Staubli VAL3: PALLET.pjx

--- PALLET.pjx ---
Parameters version=s7.5 stackSize=5000 millimeterUnit=true
Program file=back.pgx
Program file=changeOffset.pgx
Program file=changeSpeed.pgx
Program file=computeFrame.pgx
Program file=delete.pgx
Program file=deleteItem.pgx
Program file=duplicate.pgx
Program file=find.pgx
Program file=get.pgx
Program file=getDistance.pgx
Program file=getFrame.pgx
Program file=getFrameId.pgx
Program file=getFunctionEdit.pgx
Program file=getFunctionSel.pgx
Program file=getFunctionView.pgx
Program file=getListItem.pgx
Program file=getPalletData.pgx
Program file=getPalletPos.pgx
Program file=getPoint.pgx
Program file=getSize.pgx
Program file=getSizeItem.pgx
Program file=getSizePallet.pgx
Program file=getTime.pgx
Program file=getTool.pgx
Program file=getTrajItem.pgx
Program file=getTrajType.pgx
Program file=getType.pgx
Program file=goTo.pgx
Program file=HerePoint.pgx
Program file=insertItem.pgx
Program file=load.pgx
Program file=loadAction.pgx
Program file=loadCycle.pgx
Program file=loadPage.pgx
Program file=makeTraj.pgx
Program file=new.pgx
Program file=next.pgx
Program file=onEdit.pgx
Program file=onEditItem.pgx
Program file=onEditTrsf.pgx
Program file=onFunctionEdit.pgx
Program file=onFunctionSel.pgx
Program file=onFunctionView.pgx
Program file=onInsert.pgx
Program file=onProgEnd.pgx
Program file=onRun.pgx
Program file=onSave.pgx
Program file=onStart.pgx
Program file=onStop.pgx
Program file=reset.pgx
Program file=setFrameId.pgx
Program file=setPalletData.pgx
Program file=setPalletPos.pgx
Program file=setTool.pgx
Program file=setTrajItem.pgx
Program file=showTrsf.pgx
Data file=PALLET.dtx
Library alias=saveData path=Disk://saveData/saveData.pjx
Library alias=use path=Disk://kernel/userPage/userPage.pjx
Library alias=tcp path=Disk://kernel/tool/tool.pjx
Library alias=cycleStatus path=Disk://cycleStatus/cycleStatus.pjx
Library alias=pt path=Disk://kernel/template/session/saveTraj/PALLET/PALLET.pjx
Library alias=page path=Disk://kernel/template/page/page.pjx
Library alias=language path=Disk://kernel/language/language.pjx
Library alias=language2 path=Disk://trajectory/PALLET/language/language.pjx
Type name=TrajectoryItem path=Disk://kernel/template/TrajectoryItem/TrajectoryItem.pjx
Type name=ActionItem path=Disk://kernel/template/ActionItem/ActionItem.pjx
Type name=Trajectory path=Disk://kernel/template/Trajectory/Trajectory.pjx
Type name=InstrItem path=Disk://kernel/template/InstrItem/InstrItem.pjx
Type name=TrajPallet path=Disk://kernel/template/TrajPallet/TrajPallet.pjx
Type name=FrameItem path=Disk://kernel/template/FrameItem/FrameItem.pjx
Type name=ToolItem path=Disk://kernel/template/ToolItem/ToolItem.pjx

--- PALLET.dtx ---
num nOldIndex
num nStep
string sInstruction
public string sItems
string sMessage
string sMenu
public bool bMoveType[3]
  [0] = true
  [1] = true
public bool bStepping
bool bToSave
string sTrajType
Trajectory tTraj
  [0]
    TrajectoryItem tSuper
      [0]
        num distance
        num moveType
        num nTime
        num nStop
        num nTcpAction
        string comment
        bool toStop
        mdesc nom_speed = {tmax=300, rmax=9999, leave=30, reach=30}
        InstrItem iInstr[3]
          [0]
            string sType
            string sData
          [1]
            string sType
            string sData
          [2]
            string sType
            string sData
        num nMoveId
    string sID
    num nId
mdesc mMdesc = {accel=10, vel=10, blend=off}
num nKey
frame fSetFrame = {fatherId=world[0]}
TrajPallet pEditPoint
  [0]
    TrajPointItem tData
      [0]
        TrajectoryItem tSuper
          [0]
            num distance
            num moveType
            num nTime
            num nStop
            num nTcpAction
            string comment
            bool toStop
            mdesc nom_speed = {tmax=600, rmax=9999, leave=30, reach=30}
            InstrItem iInstr[3]
              [0]
                string sType
                string sData
              [1]
                string sType
                string sData
              [2]
                string sType
                string sData
            num nMoveId
        pointRx pPoint = {fatherId=pEditPoint[0].fFrame[0]}
        num nType
    frame fFrame = {fatherId=pEditPoint[0].fReference[0]}
    num nIndexTool
    string sID
    trsf trAppro[2]
    trsf trDepart[2]
    num nX = 1
    num nY = 1
    num nZ = 1
    num nIndex
    num nDistanceXYZ[3]
      [0] = 1
      [1] = 1
      [2] = 1
    string sAction
    pointRx pO = {fatherId=pEditPoint[0].fReference[0]}
    pointRx pX = {fatherId=pEditPoint[0].fReference[0]}
    pointRx pY = {fatherId=pEditPoint[0].fReference[0]}
    pointRx pZ = {fatherId=pEditPoint[0].fReference[0]}
    num nSpeedApproach = 500
    num nSpeedDepart = 500
    num nIndexFrame
    frame fReference = {fatherId=world[0]}
string sTrajCycle

--- back.pgx ---
public program back(string x_sItem)
  local num l_nValue
  local num l_nSize
begin
  // get the value
  call getPalletPos(x_sItem,l_nValue)
  call getSizePallet(x_sItem,l_nSize)
  // set the value -1
  if l_nValue>0
    call setPalletPos(x_sItem,l_nValue-1)
  else
    call setPalletPos(x_sItem,l_nSize-1)
  endIf
end

--- changeOffset.pgx ---
public program changeOffset(num& x_nOffset[])
  local num x
  local num y
  local num z
  local point l_pPoint
  local num l_nIndex
begin
  //
  // build the pallet
  //
  // compute
  for z=0 to pEditPoint.nZ-1
    for y=0 to pEditPoint.nY-1
      for x=0 to pEditPoint.nX-1
        // set all the points
        l_pPoint=pEditPoint.tData[l_nIndex].pPoint
        l_pPoint.trsf.x=l_pPoint.trsf.x+x_nOffset*x
        l_pPoint.trsf.y=l_pPoint.trsf.y+x_nOffset[1]*y
        l_pPoint.trsf.z=l_pPoint.trsf.z+x_nOffset[2]*z
        pEditPoint.tData[l_nIndex].pPoint=l_pPoint
        l_nIndex=l_nIndex+1
      endFor
    endFor
  endFor
  //
end

--- changeSpeed.pgx ---
program changeSpeed(num x_nType, num x_nIndex)
  local string l_sMessage[2]
  local num l_nActual
  local num l_nOldValue
  local num l_nSize
  local num i
begin
  //
  // change all the speed
  //
  switch x_nType
    case 0
      // APPROACH
      call language2:message(l_sMessage,0)
      call language2:message(l_sMessage[1],2)
      l_nActual=l_nOldValue=pEditPoint.nSpeedApproach
      call use:insertDialog(l_sMessage+" "+l_sMessage[1],pEditPoint.nSpeedApproach,1,6000)
    break
    case 1
      // DEPART
      call language2:message(l_sMessage,1)
      call language2:message(l_sMessage[1],2)
      l_nActual=l_nOldValue=pEditPoint.nSpeedDepart
      call use:insertDialog(l_sMessage+" "+l_sMessage[1],pEditPoint.nSpeedDepart,1,6000)
    break
    case 2
      // NORMAL SPEED
      call language:message(l_sMessage,161)
      if pEditPoint.tData[x_nIndex].tSuper.moveType==0
        l_nActual=l_nOldValue=pEditPoint.tData[x_nIndex].tSuper.nom_speed.vel
        call use:insertDialog(l_sMessage,l_nActual,1,400)
      else
        if pEditPoint.tData[x_nIndex].tSuper.moveType==1
          l_nActual=l_nOldValue=pEditPoint.tData[x_nIndex].tSuper.nom_speed.tvel
          call use:insertDialog(l_sMessage,l_nActual,1,6000)
        endIf
      endIf
    break
  endSwitch
  // set all the speed
  if l_nActual!=l_nOldValue and x_nType==2
    // normal speed, 2
    call getSizeItem(false,l_nSize)
    for i=0 to (l_nSize-1)
      if (pEditPoint.tData[i].tSuper.moveType==0)and(l_nOldValue==pEditPoint.tData[i].tSuper.nom_speed.vel)
        pEditPoint.tData[i].tSuper.nom_speed.vel=l_nActual
      else
        if (pEditPoint.tData[i].tSuper.moveType==1)and(l_nOldValue==pEditPoint.tData[i].tSuper.nom_speed.tvel)
          pEditPoint.tData[i].tSuper.nom_speed.tvel=l_nActual
        endIf
      endIf
    endFor
  endIf
  // to be saved
  bToSave=true
end

--- computeFrame.pgx ---
public program computeFrame(num x_nNewFrame)
  local num i
begin
  // recompute all the point into the new frame
  //
  for i=0 to size(pEditPoint.tData)-1
    pEditPoint.tData[i].pPoint.trsf=!pEditPoint.tData[i].pPoint.trsf*!pEditPoint.fFrame.trsf*!pEditPoint.fReference.trsf*saveData:fFrameItem[x_nNewFrame].fFrame.trsf*pEditPoint.fFrame.trsf
  endFor
  // update the reference FRAME
  pEditPoint.fReference.trsf=saveData:fFrameItem[x_nNewFrame].fFrame.trsf
end

--- deleteItem.pgx ---
public program deleteItem(num& x_nIndex)
  local num i
  local string l_sItem
begin
  // delete the selected item
  if pEditPoint.tData[x_nIndex].nType!=1 and size(pEditPoint.tData)>3
    // delete all the field
    delete(pEditPoint.tData[x_nIndex])
  else
    // not possible to delete the point
    if  pEditPoint.tData[x_nIndex].nType!=1
      pEditPoint.tData[x_nIndex].pPoint.trsf={0,0,0,0,0,0}
    endIf
    x_nIndex=-1
  endIf
end

--- duplicate.pgx ---
public program duplicate(string x_sCopy, string x_sPaste, num& x_nResult[])
  local num i
  local num l_nSize
  local string l_sItem
  local bool l_bFound
  local num l_nResult
  local string l_sString
  local num l_nX
  local num l_nY
begin
  // duplicate

  // look if the items exist
  if insert(pt:tTraj[x_sPaste])
    // link the point
    call pt:copy_it(x_sCopy,x_sPaste)
    call pt:link_all(x_sPaste)
    // save it
    bToSave=true
  endIf
end

--- get.pgx ---
public program get(string& x_sItem[], num x_nIndex)
  local string l_sKey
  local num i
  local string l_sItem
begin
  // start from the first
  l_sKey=first(pt:tTraj)
  // search it
  while l_sKey!=""
    x_sItem=l_sKey
    l_sKey=next(pt:tTraj[l_sKey])
    if i==x_nIndex
      return
    else
      i=i+1
    endIf
  endWhile
end

--- getDistance.pgx ---
public program getDistance(tool x_tTool, num& x_nDistance[], bool x_bCycle, num x_nIndex)
  local num l_nDistance
  local point l_pPoint
  local num l_nValue
  local trsf l_trsfEmpty
  local point l_pActual
  local point l_pPrev
begin
  // first point
  if x_bCycle
    // an other one
    //
    // get the point
    //
    l_pActual=pt:tTraj[sTrajCycle].tData[x_nIndex].pPoint
    // point
    x_nDistance=distance(l_pActual.trsf,pt:tTraj[sTrajCycle].trAppro[1])
  else
    l_pActual=pEditPoint.tData[x_nIndex].pPoint
    // point
    x_nDistance=distance(l_pActual.trsf,pt:tTraj[sTrajCycle].trDepart[1])
  endIf
end

--- getFrame.pgx ---
public program getFrame(frame& x_fFrame[], bool x_bCycle)
begin
  if x_bCycle
    x_fFrame.trsf=position(pt:tTraj[sTrajCycle].fFrame,world)
  else
    // update the frame
    x_fFrame.trsf=position(pEditPoint.fFrame,world)
  endIf
end

--- getFunctionEdit.pgx ---
public program getFunctionEdit(string& x_sName[])
  local string l_sMessage
begin
  //
  // define your message for the
  // function KEY
  //
  // NOTE is an ARRAY[0..7]
  //
  // example:
  // x_sName[1]="DEMO"
  // active the F2 button
  //
  // HERE
  call language:message(l_sMessage,150)
  x_sName[0]=l_sMessage
  // ALIGN
  call language:message(l_sMessage,134)
  x_sName[1]=l_sMessage
  // REACH
  call language:message(l_sMessage,152)
  x_sName[2]=l_sMessage
  // APPROACH
  call language2:message(l_sMessage,5)
  x_sName[5]=l_sMessage
  //x_sName[5]=" "
  // DEPART
  call language2:message(l_sMessage,6)
  x_sName[6]=l_sMessage
  //x_sName[6]=" "
end

--- getFunctionView.pgx ---
public program getFunctionView(string& x_sName[])
  local string l_sMessage
begin
  //
  // define your message for the
  // function KEY
  //
  // NOTE is an ARRAY[0..7]
  //
  // example:
  // x_sName[1]="DEMO"
  // active the F2 button

  // HERE
  call language:message(l_sMessage,150)
  x_sName[0]=l_sMessage
  // ALIGN
  call language:message(l_sMessage,134)
  x_sName[1]=l_sMessage
  //
  // DISABLE
  //
  // Paste
  x_sName[3]=" "
  // Mark
  x_sName[4]=" "
  // Insert
  x_sName[5]=" "
  // Delete
  x_sName[6]=" "
end

--- getListItem.pgx ---
public program getListItem(string& x_sItem[], num x_nIndex)
  local string l_sItem[12]
  local trsf l_tTrsf
  local string l_sMessage[2]
  local point l_pPoint[2]
begin
  l_pPoint=pEditPoint.tData[x_nIndex].pPoint
  l_tTrsf=l_pPoint.trsf
  l_sItem[0]=("coord  X > "+toString(".2",l_tTrsf.x))
  l_sItem[1]=("coord  Y > "+toString(".2",l_tTrsf.y))
  l_sItem[2]=("coord  Z > "+toString(".2",l_tTrsf.z))
  l_sItem[3]=("coord RX > "+toString(".2",l_tTrsf.rx))
  l_sItem[4]=("coord RY > "+toString(".2",l_tTrsf.ry))
  l_sItem[5]=("coord RZ > "+toString(".2",l_tTrsf.rz))
  // approach
  call language2:message(l_sMessage,3)
  call use:strfill(l_sMessage,8,l_sMessage)
  call showTrsf(pEditPoint.trAppro,l_sMessage[1])
  l_sItem[6]=(l_sMessage+"1>"+l_sMessage[1])
  call showTrsf(pEditPoint.trAppro[1],l_sMessage[1])
  l_sItem[7]=(l_sMessage+"2>"+l_sMessage[1])
  // approach speed
  call language2:message(l_sMessage,5)
  call use:strfill(l_sMessage,9,l_sMessage)
  l_sItem[8]=(l_sMessage+"> "+toString("",pEditPoint.nSpeedApproach))
  // depart
  call language2:message(l_sMessage,4)
  call use:strfill(l_sMessage,8,l_sMessage)
  call showTrsf(pEditPoint.trDepart,l_sMessage[1])
  l_sItem[9]=(l_sMessage+"1>"+l_sMessage[1])
  call showTrsf(pEditPoint.trDepart[1],l_sMessage[1])
  l_sItem[10]=(l_sMessage+"2>"+l_sMessage[1])
  // depart speed
  call language2:message(l_sMessage,6)
  call use:strfill(l_sMessage,9,l_sMessage)
  l_sItem[11]=(l_sMessage+"> "+toString("",pEditPoint.nSpeedDepart))
  // copy it
  call use:stringCopy(l_sItem,x_sItem)
end

--- getPalletData.pgx ---
public program getPalletData(bool x_bCycle, TrajPallet& x_tTrajPallet)
begin
  // get the Pallet DATA
  if x_bCycle
    x_tTrajPallet=pt:tTraj[sTrajCycle]
  else
    x_tTrajPallet=pEditPoint
  endIf
end

--- getPalletPos.pgx ---
public program getPalletPos(string x_sItem, num& x_nIndex[])
  local num i
  local string l_sName
  local num l_nPos
  local num l_nSize
begin
  // init the index
  x_nIndex=-1
  // scan it
  if isDefined(pt:tTraj[x_sItem])
    x_nIndex=pt:tTraj[x_sItem].nIndex
    //
  endIf
end

--- getPoint.pgx ---
public program getPoint(point& x_pPoint[], bool x_bCycle, num x_nIndex)
  local string l_sItem
begin
  // take
  if x_bCycle
    x_pPoint=pt:tTraj[sTrajCycle].tData[x_nIndex].pPoint
  else
    // give back the point
    x_pPoint=pEditPoint.tData[x_nIndex].pPoint
  endIf
end

--- getSize.pgx ---
public program getSize(num& x_nSize[])
  local string l_sType
  local string l_sKey
  local num i
  local string l_sItem
  local string l_sPath
  local num l_nResult
begin
  // give back the size
  x_nSize=size(pt:tTraj)
end

--- getSizePallet.pgx ---
public program getSizePallet(string x_sItem, num& x_nSize)
  local string l_sType
  local string l_sKey
  local num i
begin
  //
  // get the size of the collection
  //
  if isDefined(pt:tTraj[x_sItem])
    x_nSize=size(pt:tTraj[x_sItem].tData)
  else
    x_nSize=0
  endIf
end

--- getTool.pgx ---
public program getTool(num& x_nTool)
begin
  // edit one
  x_nTool=pEditPoint.nIndexTool
end

--- getTrajItem.pgx ---
public program getTrajItem(TrajectoryItem& x_tTraj[], num x_nIndex)
begin
  //
  // get all the FIELD
  //
  x_tTraj=pEditPoint.tData[x_nIndex].tSuper
end

--- getTrajType.pgx ---
program getTrajType(string& x_sTrajType[])
  local num l_nPos
  local string l_sPath
begin
  // get the trajType
  l_sPath=libPath()
  if find(l_sPath,sTrajType)==-1 or sTrajType==""
    do
      l_nPos=find(l_sPath,"/")
      if l_nPos==-1
        l_nPos=find(l_sPath,"\")
      endIf
      if l_nPos!=-1
        l_sPath=right(l_sPath,len(l_sPath)-l_nPos-1)
      endIf
    until l_nPos==-1
    //
    sTrajType=l_sPath
  endIf
  // return back
  x_sTrajType=sTrajType
end

--- getType.pgx ---
public program getType(num& x_nType, bool x_bCycle, num x_nIndex)
begin
  // get the point Type
  if x_bCycle
    x_nType=pt:tTraj[sTrajCycle].tData[x_nIndex].nType
  else
    x_nType=pEditPoint.tData[x_nIndex].nType
  endIf
end

--- goTo.pgx ---
public program goTo(tool x_tTool, mdesc x_mDesc, num x_nMoveType, bool& x_bUnreached[], num x_nIndex)
  local string l_sMessage
  local num i
  local point l_pPoint
  local joint l_jJoint
begin
  // the maximum size
  x_mDesc.blend=off
  // get the point
  call getPoint(l_pPoint,false,x_nIndex)
  //
  // step by step motion
  //
  // go to the appro
  for i=0 to size(pEditPoint.trAppro)-1
    if !pointToJoint(x_tTool,herej(),appro(l_pPoint,pEditPoint.trAppro[i]),l_jJoint)
      // not reachable
      call language:message(l_sMessage,169)
      popUpMsg(l_sMessage)
      return
    else
      if x_nMoveType==0 and i==0
        // or is not in range
        movej(appro(l_pPoint,pEditPoint.trAppro[i]),x_tTool,x_mDesc)
      else
        movel(appro(l_pPoint,pEditPoint.trAppro[i]),x_tTool,x_mDesc)
      endIf
    endIf
  endFor
  // wait to catch the point
  wait(isEmpty() or isKeyPressed(255) or cycleStatus:nWorkingStatus!=0)
  if isEmpty()
    delay(1)
    // go directly to the point is the robot is nearby the point
    if !pointToJoint(x_tTool,herej(),l_pPoint,l_jJoint)
      // not reachable
      call language:message(l_sMessage,169)
      popUpMsg(l_sMessage)
      return
    else
      movel(l_pPoint,x_tTool,x_mDesc)
      wait(isEmpty() or isKeyPressed(255) or cycleStatus:nWorkingStatus!=0)
      if isEmpty()
        delay(1)
        // go to the depart
        for i=0 to size(pEditPoint.trDepart)-1
          if !pointToJoint(x_tTool,herej(),appro(l_pPoint,pEditPoint.trDepart[i]),l_jJoint)
            // not reachable
            call language:message(l_sMessage,169)
            popUpMsg(l_sMessage)
            return
          else
            movel(appro(l_pPoint,pEditPoint.trDepart[i]),x_tTool,x_mDesc)
          endIf
        endFor
        wait(isEmpty() or isKeyPressed(255) or cycleStatus:nWorkingStatus!=0)
      endIf
    endIf
  endIf
end

--- HerePoint.pgx ---
public program HerePoint(num x_nIndex)
  local tool l_tTool
  local point l_pHere
  local frame l_fFrame
  local num i
  local num l_nIndex
  local num l_nSize
begin
  //
  // take the point
  //
  // tool
  call tcp:getTool(l_tTool,pEditPoint.nIndexTool)
  // here
  l_pHere=here(l_tTool,pEditPoint.fFrame)
  resetMotion()
  // save the trsf
  pEditPoint.tData[x_nIndex].pPoint.trsf=l_pHere.trsf
  // check the moveType to save the config
  if pEditPoint.tData[x_nIndex].tSuper.moveType==0
    pEditPoint.tData[x_nIndex].pPoint.config=l_pHere.config
  endIf
end

--- insertItem.pgx ---
public program insertItem(num& x_nIndexCopy, num x_nIndexPaste)
  local num l_nLastType
  local point l_pPoint
  local num l_nType
begin
  //
  // use to add more elements from the typical one
  //
  // insert all the field
  //
  l_pPoint=pEditPoint.tData[x_nIndexCopy].pPoint
  link(pEditPoint.tData[x_nIndexPaste].pPoint,pEditPoint.fFrame)
  insert(pEditPoint.tData[x_nIndexPaste])
  // set IT
  pEditPoint.tData[x_nIndexPaste].pPoint.trsf=l_pPoint.trsf
end

--- load.pgx ---
public program load(string x_sItem, num& x_nResult)
  local string l_sType
  local string l_sMessage
  local num i
  local num l_nResult
begin
  // load the select trajectory..already loaded
  call getTrajType(l_sType)
  if find(pt:libPath(),saveData:sPathTraj)==-1
    l_nResult=pt:libLoad(saveData:sPathTraj+l_sType)
    delay(0)
    if saveData:bDebug or l_nResult!=0
      ? "loading PALLET..."+saveData:sPathTraj+l_sType + toString("",l_nResult)
    endIf
  endIf
  // use the type...
  if isDefined(pt:tTraj[x_sItem])
    call pt:link_all(x_sItem)
    pEditPoint=pt:tTraj[x_sItem]
    pEditPoint.sID=x_sItem
    link(pEditPoint.fReference,world)
    link(pEditPoint.fFrame,pEditPoint.fReference)
  elseIf x_sItem!=""
    // not FOUND
    call language:message(l_sMessage,-7)
    x_nResult=-1
    popUpMsg(l_sMessage+x_sItem)
    pEditPoint.sID=""
  endIf
end

--- loadAction.pgx ---
program loadAction(string x_sPallet, num x_nOffset)
  local num l_nPos
  local num l_nSize[3]
  local string l_sAction
begin
  //
  // get the actual position
  //
  call getPalletPos(x_sPallet,l_nPos)
  // PLANE CONDITION
  // loook for the z quote
  l_sAction=pt:tTraj[sTrajCycle].sAction[l_nPos%pt:tTraj[sTrajCycle].nZ]
  if (l_nPos+1)%(pt:tTraj[sTrajCycle].nY*pt:tTraj[sTrajCycle].nX)==0 and l_sAction!=""
    // show the string
    cycleStatus:sToShow="CALL PALLET PROG "+l_sAction
    // SET THE JUMP for the CALL..
    cycleStatus:bCALL=true
    // NB use the session field
    cycleStatus:iToSuperV.sType="PROG"
    cycleStatus:iToSuperV.sData=l_sAction
    use:bUseRefresh=true
  endIf
end

--- loadCycle.pgx ---
public program loadCycle(string x_sItem, num& x_nResult[])
  local string l_sType
  local string l_sMessage
begin
  // load the select trajectory..already loaded
  call getTrajType(l_sType)
  if find(pt:libPath(),saveData:sPathTraj)==-1
    pt:libLoad(saveData:sPathTraj+l_sType)
    delay(0)
    if saveData:bDebug
      ? "loading PALLET..."+saveData:sPathTraj+l_sType
    endIf
  endIf
  if isDefined(pt:tTraj[x_sItem])
    call pt:link_all(x_sItem)
    // use the type...
    sTrajCycle=x_sItem
  else
    // not FOUND
    call language:message(l_sMessage,-7)
    x_nResult=-1
    cycleStatus:bToStop=true
    popUpMsg(l_sMessage+x_sItem)
  endIf
end

--- loadPage.pgx ---
program loadPage(string x_sPage, string& x_sItems[])
// load the next page
  local num i
  local string l_sMessage
begin
  // look if the page libload is correct
  i=page:libLoad(x_sPage)
  delay(0)
  if i!=0
    logMsg("[KERNEL] INTERFACE:PAGE LIBLOAD "+x_sPage+" result "+toString("",i))
    call language:message(l_sMessage,-7)
    popUpMsg(l_sMessage+x_sPage+" ; "+toString("",i))
  else
    // copy all the field from x_sItems to the next page
    call use:stringCopy(x_sItems,page:sItems)
    call page:main()
    // to give back
    call use:stringCopy(page:sItems,x_sItems)
  endIf
end

--- makeTraj.pgx ---
public program makeTraj(string& x_sItem[])
  local num i
  local num l_nDistance
  local num l_nSize
  local tool l_tTool
  local num l_nMoveId
  local point l_pPoint
  local string l_sType
  local TrajectoryItem l_tTraj
  local ActionItem l_aAction
  local num l_nIndex
  local mdesc l_nomSpeed
begin
  // take the TOOL
  call tcp:getTool(l_tTool,pt:tTraj[sTrajCycle].nIndexTool)
  // the maximum size
  call getSizeItem(true,l_nSize)
  //
  // for all of my traj cyclePoints move the robot
  //
  // one element
  resize(tTraj.tSuper,1,1)
  tTraj.tSuper=pt:tTraj[sTrajCycle].tData[pt:tTraj[sTrajCycle].nIndex].tSuper
  tTraj.tSuper.comment="["+toString("2",pt:tTraj[sTrajCycle].nIndex+1)+"/"+toString("2",size(pt:tTraj[sTrajCycle].tData))+"] "+tTraj.tSuper.comment
  tTraj.sID="PALLET "+pt:tTraj[sTrajCycle].sID
  call cycleStatus:addTraj(tTraj)
  //
  // get the point info
  //
  l_nIndex=pt:tTraj[sTrajCycle].nIndex
  l_tTraj=pt:tTraj[sTrajCycle].tData[l_nIndex].tSuper
  call getPoint(l_pPoint,true,l_nIndex)
  //
  // put the move in the stack
  //
  // go to the appro
  for i=0 to size(pt:tTraj[sTrajCycle].trAppro)-1
    if l_tTraj.moveType==0 and i==0
      // or is not in range
      movej(appro(l_pPoint,pt:tTraj[sTrajCycle].trAppro[i]),l_tTool,l_tTraj.nom_speed)
    elseIf i==0
      movel(appro(l_pPoint,pt:tTraj[sTrajCycle].trAppro[i]),l_tTool,l_tTraj.nom_speed)
    elseIf i>0 and pt:tTraj[sTrajCycle].trAppro[i]!=pt:tTraj[sTrajCycle].trAppro[i-1]
      l_nomSpeed=l_tTraj.nom_speed
      l_nomSpeed.tvel=pt:tTraj[sTrajCycle].nSpeedApproach
      l_nomSpeed.leave=l_nomSpeed.reach=5
      movel(appro(l_pPoint,pt:tTraj[sTrajCycle].trAppro[i]),l_tTool,l_nomSpeed)
    endIf
  endFor
  //
  // get the distance in percentage
  call getDistance(l_tTool,l_nDistance,true,l_nIndex)
  //
  // give to the traj library the percentage distance
  //
  if l_tTraj.toStop
    l_tTraj.nom_speed.blend=off
  endIf
  // send the action information to cycle
  l_tTraj.nom_speed.tvel=pt:tTraj[sTrajCycle].nSpeedDepart
  l_nMoveId=movel(l_pPoint,l_tTool,l_tTraj.nom_speed)
  l_aAction.nDistance=l_nDistance
  l_aAction.nPointId=0
  l_aAction.nMoveId=l_nMoveId
  l_aAction.sIdTraj="PALLET "+pt:tTraj[sTrajCycle].sID
  call cycleStatus:putInstr_Traj(l_aAction,l_tTraj,pt:tTraj[sTrajCycle].nIndexTool,1)
  // there is a waitEndMove
  if l_tTraj.toStop
    waitEndMove()
    delay(l_tTraj.nStop)
    // wait all the action has been done
    wait(cycleStatus:bActionRunning==false)
  endIf
  // update
  l_tTraj=pt:tTraj[sTrajCycle].tData[l_nIndex].tSuper
  //  depart
  for i=0 to size(pt:tTraj[sTrajCycle].trDepart)-1
    l_nomSpeed=l_tTraj.nom_speed
    l_nomSpeed.tvel=pt:tTraj[sTrajCycle].nSpeedDepart
    if pt:tTraj[sTrajCycle].trDepart[0]!=pt:tTraj[sTrajCycle].trDepart[1]
      l_nomSpeed.leave=l_nomSpeed.reach=5
    endIf
    movel(appro(l_pPoint,pt:tTraj[sTrajCycle].trDepart[i]),l_tTool,l_nomSpeed)
  endFor
  // calculate the offset
  l_nDistance=distance(l_pPoint,appro(l_pPoint,pt:tTraj[sTrajCycle].trDepart[i-1]))
  // use a 10 % of tollerance
  if l_nDistance!=0
    l_nDistance=1-l_tTraj.nom_speed.leave/l_nDistance-0.1
  else
    l_nDistance=1-0.1
  endIf
  //
  // ACTION AFTER MOVE
  //
  call loadAction(x_sItem,l_nDistance)
end

--- next.pgx ---
public program next(string x_sItem)
  local num l_nValue
  local num l_nSize
begin
  // get the actual position
  call getPalletPos(x_sItem,l_nValue)
  call getSizePallet(x_sItem,l_nSize)
  // go to the next ONE
  if l_nValue<l_nSize-1
    call setPalletPos(x_sItem,l_nValue+1)
  else
    call setPalletPos(x_sItem,0)
  endIf
end

--- onEdit.pgx ---
public program onEdit(string& x_sItem[])
  local string l_sPath
  local num i
  local string l_sItem
  local num l_nSize
  local num l_nResult
begin
  // DEFINE YOUR ITEM
  call getTrajType(saveData:sTrajTypeUsing)
  // load the trajectory
  call load(x_sItem,l_nResult)
  if find(x_sItem,"@")==-1
    // load the page viewTraj
    l_sPath="Disk://trajectory/PALLET/page_pallet"
    // give back the path
    x_sItem[1]=x_sItem
    x_sItem=l_sPath
  endIf
end

--- onEditItem.pgx ---
public program onEditItem(string& x_sEvent[], num x_nIndex, num x_nIndexItem)
  local bool l_bReachable
  local num i
  local trsf l_tApproach[2]
  local trsf l_tDepart[2]
  local num l_nSpeed
  local string l_sMessage
  local num l_nOffset
  local string l_sMessage2
  local string l_sItem
begin
  // edit the custom element that was add in the list
  if x_nIndex<6
    // edit the TRSF
    call onEditTrsf(x_nIndex,x_nIndexItem,x_sEvent)
  else
    // i=find(x_sEvent,">")+1
    call use:findPos(x_sEvent,">",i)
    i=i+1
    call language2:message(l_sMessage2,42)
    //
    switch x_nIndex
      case 6
        // change the approach 1
        call language2:message(l_sMessage,3)
        call use:changeTrsf(pEditPoint.trAppro,l_sMessage+" [1]",l_sMessage2)
      break
      case 7
        // change the approach 2
        call language2:message(l_sMessage,3)
        call use:changeTrsf(pEditPoint.trAppro[1],l_sMessage+" [2]",l_sMessage2)
      break
      case 8
        // change the approach speed
        call use:listcursor(use:nView,false)
        l_sItem=""
        call use:changeValue(pEditPoint.nSpeedApproach,1,2000,i+40-use:nBottomX,use:nView+1,l_sItem)
      break
      case 9
        // change the depart
        call language2:message(l_sMessage,4)
        call use:changeTrsf(pEditPoint.trDepart,l_sMessage+" [1]",l_sMessage2)
      break
      case 10
        // change the depart 2
        call language2:message(l_sMessage,4)
        call use:changeTrsf(pEditPoint.trDepart[1],l_sMessage+" [2]",l_sMessage2)
      break
      case 11
        // change the depart speed
        call use:listcursor(use:nView,false)
        l_sItem=""
        call use:changeValue(pEditPoint.nSpeedDepart,1,2000,i+40-use:nBottomX,use:nView+1,l_sItem)
      break
    endSwitch
  endIf
  //
end

--- onEditTrsf.pgx ---
public program onEditTrsf(num x_nIndex, num x_nIndexItem, string x_sEvent)
  local num i
  local num l_nMin
  local num l_nMax
  local trsf l_tTrsf
  local string l_sEmpty
  local joint l_jJoint
  local tool l_tTool
  local string l_sMessage
  local trsf l_OldTrsf
begin
  // edit TRSF OF THE POINT
  l_tTrsf=pEditPoint.tData[x_nIndexItem].pPoint.trsf
  // find the >
  call use:findPos(x_sEvent,">",i)
  i=i+1
  // find the line
  if !cycleStatus:bCycle
    l_nMin=l_nMax=0
  else
    switch x_nIndex
      case 0
        // x
        l_nMin=l_tTrsf.x-10
        l_nMax=l_tTrsf.x+10
      break
      case 1
        // y
        l_nMin=l_tTrsf.y-10
        l_nMax=l_tTrsf.y+10
      break
      case 2
        // z
        l_nMin=l_tTrsf.z-10
        l_nMax=l_tTrsf.z+10
      break
      case 3
        // rx
        l_nMin=l_tTrsf.rx-5
        l_nMax=l_tTrsf.rx+5
      break
      case 4
        // ry
        l_nMin=l_tTrsf.ry-5
        l_nMax=l_tTrsf.ry+5
      break
      case 5
        // rz
        l_nMin=l_tTrsf.rz-5
        l_nMax=l_tTrsf.rz+5
      break
    endSwitch
  endIf
  // clean the line
  call use:listcursor(use:nView,false)
  //
  switch x_nIndex
    case 0
      //  x-value
      call use:changeValue(l_tTrsf.x,l_nMin,l_nMax,i+40-use:nBottomX,use:nView+1,l_sEmpty)
    break
    case 1
      //  y-value
      call use:changeValue(l_tTrsf.y,l_nMin,l_nMax,i+40-use:nBottomX,use:nView+1,l_sEmpty)
    break
    case 2
      //  z-value
      call use:changeValue(l_tTrsf.z,l_nMin,l_nMax,i+40-use:nBottomX,use:nView+1,l_sEmpty)
    break
    case 3
      //  rx-value
      call use:changeValue(l_tTrsf.rx,l_nMin,l_nMax,i+40-use:nBottomX,use:nView+1,l_sEmpty)
    break
    case 4
      //  ry-value
      call use:changeValue(l_tTrsf.ry,l_nMin,l_nMax,i+40-use:nBottomX,use:nView+1,l_sEmpty)
    break
    case 5
      //  rz-value
      call use:changeValue(l_tTrsf.rz,l_nMin,l_nMax,i+40-use:nBottomX,use:nView+1,l_sEmpty)
    break
  endSwitch
  // validate
  if !use:bUseEscape
    // check the config
    l_tTool=saveData:tData[pEditPoint.nIndexTool].tcp
    l_OldTrsf=pEditPoint.tData[x_nIndexItem].pPoint.trsf
    pEditPoint.tData[x_nIndexItem].pPoint.trsf=l_tTrsf
    if !pointToJoint(l_tTool,herej(),pEditPoint.tData[x_nIndexItem].pPoint,l_jJoint)
      // not reachable
      pEditPoint.tData[x_nIndexItem].pPoint.trsf=l_OldTrsf
      call language:message(l_sMessage,169)
      popUpMsg(l_sMessage)
    endIf
  endIf
end

--- onFunctionEdit.pgx ---
public program onFunctionEdit(num x_nIndex, string x_sEvent, num x_nFunctionKey)
  local string l_sMessage
  local string l_sButton[2]
  local bool l_bOk
  local string l_sPage
  local string l_sItem
  local tool l_tTool
  local point l_pAlign
  local bool l_bYes
  local string l_sMessage2
begin
  //
  // do on Key action
  //
  // x_nIndex = actual index item
  // x_sEvent = actual event item
  //
  switch x_nFunctionKey
    // F1 button
    case 271
      // HERE POINT
      if !cycleStatus:bCycle
        call language:message(l_sMessage,160)
        call language:getYesNo(l_sButton)
        call use:yes_no(l_sMessage,l_sButton,l_bOk)
        if l_bOk
          call HerePoint(x_nIndex)
        endIf
      endIf
    break
    // F2 button
    case 272
      // ALIGN
      if !cycleStatus:bCycle
        resetMotion()
        call getFrame(fSetFrame,false)
        // tool
        call tcp:getTool(l_tTool,pEditPoint.nIndexTool)
        l_pAlign=here(l_tTool,world)
        l_pAlign.trsf=align(l_pAlign.trsf,fSetFrame.trsf)
        call language:message(l_sMessage,203)
        call language:message(l_sMessage2,134)
        l_sMessage=l_sMessage+" "+l_sMessage2+"..."
        call use:timerDialog(l_sMessage,0)
        movej(l_pAlign,l_tTool,mMdesc)
        watch(isEmpty() or isKeyPressed(255),3)
        if !isEmpty()
          resetMotion()
        endIf
        delay(2)
      endIf
    break
    // F3 button
    case 273
      // Select the gun
      l_sPage="Disk://kernel/page/tool"
      call loadPage(l_sPage,l_sItem)
      // set the tool
      pEditPoint.nIndexTool=saveData:nIndexTool
    break
    // F4 button
    case 274
    break
    // F5 button
    case 275
    break
    // F6 button
    case 276
      // change all the approach speed
      call changeSpeed(0,x_nIndex)
    break
    // F7 button
    case 277
      // change all the depart speed
      call changeSpeed(1,x_nIndex)
    break
    // F8 button
    case 278
      // save it
      bToSave=true
    break
  endSwitch
end

--- onFunctionSel.pgx ---
public program onFunctionSel(num x_nIndex, string x_sEvent, num x_nFunctionKey)
begin
  //
  // do on Key action
  //
  // x_nIndex = actual index item
  // x_sEvent = actual event item
  //
  switch x_nFunctionKey
    // F1 button
    case 271
    break
    // F2 button
    case 272
    break
    // F3 button
    case 273
    break
    // F4 button
    case 274
    break
    // F5 button
    case 275
    break
    // F6 button
    case 276
    break
    // F7 button
    case 277
    break
    // F8 button
    case 278
    break
  endSwitch
end

--- onFunctionView.pgx ---
public program onFunctionView(num x_nIndex, string x_sEvent, num x_nFunctionKey)
  local string l_sMessage
  local string l_sButton[2]
  local bool l_bOk
  local tool l_tTool
  local point l_pAlign
  local string l_sMessage2
  local joint l_jJoint
begin
  //
  // do on Key action
  //
  // x_nIndex = actual index item
  // x_sEvent = actual event item
  //
  switch x_nFunctionKey
    case 271
      // HERE POINT
      if !cycleStatus:bCycle
        call language:message(l_sMessage,160)
        call language:getYesNo(l_sButton)
        call use:yes_no(l_sMessage,l_sButton,l_bOk)
        if l_bOk
          call HerePoint(x_nIndex)
        endIf
      endIf
    break
    // F2 button
    case 272
      // ALIGN
      if !cycleStatus:bCycle and !cycleStatus:bSimulation
        resetMotion()
        call getFrame(fSetFrame,false)
        // tool
        call tcp:getTool(l_tTool,pEditPoint.nIndexTool)
        l_pAlign=here(l_tTool,world)
        l_pAlign.trsf=align(l_pAlign.trsf,fSetFrame.trsf)
        // check the align
        if pointToJoint(l_tTool,herej(),l_pAlign,l_jJoint)
          call language:message(l_sMessage,203)
          call language:message(l_sMessage2,134)
          l_sMessage=l_sMessage+" "+l_sMessage2+"..."
          call use:timerDialog(l_sMessage,0)
          movel(l_pAlign,l_tTool,mMdesc)
          watch(isEmpty() or isKeyPressed(255),3)
          if !isEmpty()
            resetMotion()
          endIf
          delay(2)
        endIf
      endIf
    break
    // F3 button
    case 273
    break
    // F4 button
    case 274
    break
    // F5 button
    case 275
    break
    // F6 button
    case 276
    break
    // F7 button
    case 277
    break
    // F8 button
    case 278
    break
  endSwitch
end

--- onInsert.pgx ---
public program onInsert(string& x_sItem[])
  local string l_sEvent
  local num l_nKey
  local num l_nIndex
  local num l_nSize
  local num i
  local string l_sMessage
  local bool l_bFound
  local string l_sType
  local bool l_bUseFilter
  local string l_sPaste
  local num l_nResult
  local num l_nX
  local num l_nY
  local string l_sName
begin
  // get the type
  call getTrajType(x_sItem)
  saveData:sTrajTypeUsing=x_sItem
  cls()
  // is a filter using ??
  if saveData:sTrajFilter!=""
    l_bUseFilter=true
    call language:message(l_sMessage,64)
    call use:type(0,1,l_sMessage+">ON")
  else
    // clean
    call use:typeLen(0,1," ",use:nBottomX)
  endIf
  //
  // CREATE THE LIST
  //
  // define your list size for default
  call use:setSizeList(19,0,19,11)
  call use:setView(false)
  call use:listcreate(x_sItem)
  // take the coordinate....
  l_nX=40-use:nBottomX-1
  l_nY=use:nBottomY+1
  // show the message
  call language:message(l_sMessage,61)
  call use:stringToArray(l_sMessage,sMenu)
  call use:setMenu(sMenu,true,3)
  // Build the list
  call getSize(l_nSize)
  for i=0 to l_nSize-1
    call get(l_sEvent,i)
    if l_sEvent!=""
      //
      // use the filter ?
      //
      // check if the bProcessList filter is active
      //
      l_bFound=true
      if saveData:sTrajFilter!=""
        l_bFound=find(l_sEvent,saveData:sTrajFilter)!=-1
      endIf
      // add
      if l_bFound
        call use:listadd(l_sEvent)
      endIf
    endIf
  endFor
  call use:listupdate(0)
  do
    // get the item
    l_nKey=get()
    call use:listevent(l_nKey,l_nIndex,l_sEvent)
    if l_nKey==271 and l_bUseFilter
      // Build the list
      call getSize(l_nSize)
      // empty and rebuild
      call use:listempty()
      for i=0 to l_nSize-1
        call get(l_sEvent,i)
        if l_sEvent!=""
          call use:listadd(l_sEvent)
        endIf
      endFor
      // clean
      call use:typeLen(0,1," ",use:nBottomX)
      call use:typeMenu(1," ")
      l_bUseFilter=false
      call use:listupdate(0)
    endIf
        //
  until l_nKey==270 or l_nKey==255 or l_nKey==278 or l_nKey==276
  //
  switch l_nKey
    case 270
      // save the name
      l_sName=l_sEvent
    break
    case 276
      // duplicate
      // ask for the new
      call language:message(l_sMessage,21)
      call use:type(l_nX,l_nY,l_sMessage)
      l_sName=l_sEvent
      // read the new trajectory
      call use:read(l_nX+len(l_sMessage),l_nY,l_sName,10,false)
      if !use:bUseEscape
        call duplicate(l_sEvent,l_sName,l_nResult)
      endIf
    break
    case 278
      call language:message(l_sMessage,21)
      call use:type(l_nX,l_nY,l_sMessage)
      // read the new trajectory
      call use:read(l_nX+len(l_sMessage),l_nY,l_sName,10,false)
      if !use:bUseEscape
        // look if the items exist
        call new(l_sName,l_nResult)
        if l_nResult==-1
          call language:message(l_sMessage,-2)
          popUpMsg(l_sMessage)
        endIf
      endIf
    break
  endSwitch
  if l_nKey!=255
    x_sItem=l_sName
  else
    x_sItem=""
  endIf
end

--- onRun.pgx ---
public program onRun(string& x_sItem[])
  local string l_sEmpty
  local num l_nResult
begin
  // execute check if need to reload
  call loadCycle(x_sItem,l_nResult)
  // execute
  call makeTraj(x_sItem)
  // increase by one
  call next(x_sItem)
end

--- onSave.pgx ---
public program onSave(string& x_sItem[])
  local num i
  local num l_nSize
  local num l_nIndex
begin
  //if bToSave
  // update
  if isDefined(pt:tTraj[pEditPoint.sID])
    // to prevent error on the executing update the nIndex
    pEditPoint.nIndex=pt:tTraj[pEditPoint.sID].nIndex
    // copy the value
    pt:tTraj[pEditPoint.sID]=pEditPoint
    // link the frame
    call pt:link_all(pEditPoint.sID)
  endIf
  // saveIt
  pt:libSave()
  bToSave=false
  //endIf
end

--- onStart.pgx ---
public program onStart(string& x_sItem[])
  local num i
  local string l_sType
  local string l_sPath
begin
  call language2:getLanguage(l_sPath)
  if l_sPath!=language2:libPath()+"/"+saveData:language
    // set language
    call language2:setLanguage(language2:libPath()+"/"+saveData:language)
  endIf
  // reset all the pallet
  call reset()
end

--- onStop.pgx ---
public program onStop(string& x_sItem[])
begin
  if x_sItem=="kill"
    pt:libLoad("Disk://kernel/template/session/saveTraj/PALLET")
  endIf
end

--- reset.pgx ---
public program reset()
  local num i
  local string l_sName
  local num l_nPos
  local string l_sKey
begin
  // scan it
  l_sKey=first(pt:tTraj)
  while l_sKey!=""
    if l_sKey!=""
      pt:tTraj[l_sKey].nIndex=0
    endIf
    l_sKey=next(pt:tTraj[l_sKey])
  endWhile
  // exit
end

--- setFrameId.pgx ---
public program setFrameId(num x_nIndex)
  local num i
begin
  // save the FrameId
  pEditPoint.nIndexFrame=x_nIndex
  // link to the father frame
  pEditPoint.fReference.trsf=saveData:fFrameItem[x_nIndex].fFrame.trsf
  link(pEditPoint.fReference,world)
  link(pEditPoint.fFrame,pEditPoint.fReference)
  // link the frame and all the points
  for i=0 to size(pEditPoint.tData)-1
    link(pEditPoint.tData[i].pPoint,pEditPoint.fFrame)
  endFor
end

--- setPalletData.pgx ---
public program setPalletData(TrajPallet& x_tTrajPallet)
  local num i
begin
  // set the Pallet DATA
  pEditPoint=x_tTrajPallet
  // link it
  for i=0 to size(pEditPoint.tData)-1
    link(pEditPoint.tData[i].pPoint,pEditPoint.fFrame)
  endFor
end

--- setPalletPos.pgx ---
public program setPalletPos(string x_sItem, num x_nValue)
  local num i
  local string l_sName
  local num l_nPos
begin
  // scan it
  if isDefined(pt:tTraj[x_sItem])
    // redefine the position
    pt:tTraj[x_sItem].nIndex=x_nValue
  endIf
end

--- setTool.pgx ---
public program setTool(num x_nIndexTool)
begin
  // set the TOOL
  pEditPoint.nIndexTool=x_nIndexTool
end

--- showTrsf.pgx ---
program showTrsf(trsf x_tTrsf, string& x_sTrsf[])
begin
  x_sTrsf="("+toString("",x_tTrsf.x)+","+toString("",x_tTrsf.y)+","+toString("",x_tTrsf.z)+","+toString("",x_tTrsf.rx)+","+toString("",x_tTrsf.ry)+","+toString("",x_tTrsf.rz)+")"
end
